TYPE MachiningStation_Coils :
STRUCT
	EStop_Out			: BOOL;
	Part_Reset			: BOOL;
	Robot_Proximity		: BOOL;
	Kill_Simulator		: BOOL;
END_STRUCT
END_TYPE

(* stored: Version 1.1.0.1, ProductVersion 3.1.0.36
   DUT MachiningStation_Coils: Id {b7324d07-6856-4b64-8ffd-a2b5959f0c63} *)
